VISUALIZATION Visualization  // 2x2
END_VISUALIZATION

(* stored: Version 1.1.0.1, ProductVersion 3.1.4022.10
   Visu Visualization: Id {92f9d153-1cef-4734-8fee-1331a5a6485c} *)
